SUBAPPLICATION WBSD_Auswahl (* Waehlt per Button die radbasierte Geschwindigkeit/Distanz (WBSD) als Quelle aus, merkt sich die Auswahl persistent im NVS, setzt bei Auswahl die anderen Quellen zurueck und liefert die WBSD-Sensordaten nach aussen *)
  (* Standard: 61499-2 *)
  (* Version 1.0, 2026-08-27, Franz *)
  PACKAGE FBs::Baumsetzer::func::Automatik;
  IMPORT NVS_Keys::Key_WBSD_Store;
  IMPORT isobus::UT::io::Button::ButtonActivationCode::BT_RELEASED_UNLATCHED;
  IMPORT test::FBs::Baumsetzer::Constants::DefaultPool::Button_WBSD;
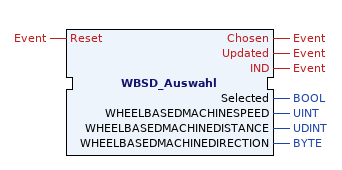
  EVENT_INPUT
    Reset; (* Anforderung von einer der anderen Quellen: eigene Auswahl zuruecksetzen *)
  END_EVENT
  EVENT_OUTPUT
    Chosen; (* Button_WBSD wurde gedrueckt: eigene Auswahl setzen und alle anderen Quellen zuruecksetzen *)
    Updated; (* Ausgewaehlt-Status verfuegbar bzw. geaendert (Init-Lesen oder Aenderung); Trigger fuer nachgelagerte Verarbeitung (u.a. Hintergrundfarbe) *)
    IND; (* Neue WBSD-Daten empfangen (Indication von I_WBSD) *)
  END_EVENT
  VAR_OUTPUT
    Selected : BOOL; (* TRUE wenn WBSD aktuell als Geschwindigkeitsquelle ausgewaehlt ist *)
    WHEELBASEDMACHINESPEED : UINT; (* Radbasierte Maschinengeschwindigkeit (PGN 65096, SPN 1862) *)
    WHEELBASEDMACHINEDISTANCE : UDINT; (* Radbasierte Maschinendistanz (PGN 65096, SPN 1863) *)
    WHEELBASEDMACHINEDIRECTION : BYTE; (* Radbasierte Fahrtrichtung (PGN 65096, SPN 1864) *)
  END_VAR
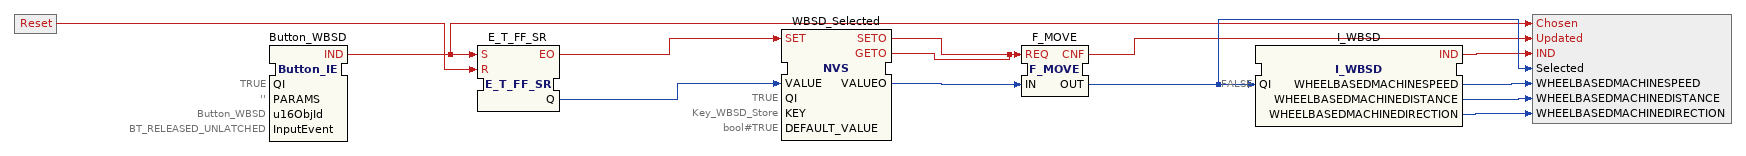
  FBS
    Button_WBSD : isobus::UT::io::Button::Button_IE(QI := TRUE, PARAMS := '', u16ObjId := Button_WBSD, InputEvent := BT_RELEASED_UNLATCHED);
    E_T_FF_SR : iec61499::events::E_T_FF_SR;
    WBSD_Selected : logiBUS::storage::esp32_nvs::NVS(QI := TRUE, KEY := Key_WBSD_Store, DEFAULT_VALUE := bool#TRUE);
    F_MOVE : iec61131::selection::F_MOVE; {SET_ATTRIBUTE(DataType, BOOL)}
    I_WBSD : isobus::tecu::I_WBSD(QI := FALSE);
  END_FBS
  EVENT_CONNECTIONS
    Button_WBSD.IND TO E_T_FF_SR.S;
    Button_WBSD.IND TO Chosen;
    Reset TO E_T_FF_SR.R;
    E_T_FF_SR.EO TO WBSD_Selected.SET;
    WBSD_Selected.SETO TO F_MOVE.REQ;
    WBSD_Selected.GETO TO F_MOVE.REQ;
    F_MOVE.CNF TO Updated;
    I_WBSD.IND TO IND;
  END_CONNECTIONS
  DATA_CONNECTIONS
    E_T_FF_SR.Q TO WBSD_Selected.VALUE;
    WBSD_Selected.VALUEO TO F_MOVE.IN;
    F_MOVE.OUT TO I_WBSD.QI;
    F_MOVE.OUT TO Selected;
    I_WBSD.WHEELBASEDMACHINESPEED TO WHEELBASEDMACHINESPEED;
    I_WBSD.WHEELBASEDMACHINEDISTANCE TO WHEELBASEDMACHINEDISTANCE;
    I_WBSD.WHEELBASEDMACHINEDIRECTION TO WHEELBASEDMACHINEDIRECTION;
  END_CONNECTIONS
END_SUBAPPLICATION
